{attribute 'qualified_only'}
VAR_GLOBAL
	_SAVED_DATA : ARRAY[1..PARAM_MOTION_SAVEPOINT.SUPPORTED_SLOTS] OF S_SAVEPOINT;
END_VAR

(* stored: Version 1.1.0.1, ProductVersion 3.1.4019.2
   GVL GVL_MOTION_SAVEPOINT: Id {543a84c2-71f1-44b6-b817-43093ebfb87f} *)
